Staubli VAL3: deleteItem.pgx

public program deleteItem(num& x_nIndex)
  local num i
  local string l_sItem
begin
  // delete the selected item
    // delete all the field
    delete(pEditPoint.tData[x_nIndex])
end
